Staubli VAL3: stringCopy.pgx

public program stringCopy(string& x_sCopy[], string& x_sPaste[])
// Copy all the value from the x_sCopy to x_sPaste
  local num i
  local num l_nSize
begin
  // Copy all the value from the first element to the second one
  //
  // redim the Paste String ARRAY
  //
  l_nSize=size(x_sPaste)
  if size(x_sCopy)>size(x_sPaste)
    for i=l_nSize to (size(x_sCopy)-1)
      $dins(x_sPaste,i)
    endFor
  else
    if size(x_sCopy)<size(x_sPaste)
      for i=size(x_sCopy) to l_nSize-1
        $ddel(x_sPaste,size(x_sCopy))
      endFor
    endIf
  endIf
  // COPY ALL THE FIELD
  for i=0 to (size(x_sCopy)-1)
    x_sPaste[i]=x_sCopy[i]
  endFor
end
